FUNCTION_BLOCK TagCmp IMPLEMENTS I_TagCmp
VAR
	_iBaseTag		: I_Tag;
	_eResult		: Results.Result;
	_bLock			: BOOL;
END_VAR

PROPERTY PRIVATE _self : I_TagCmp
GET
VAR
	_this : I_TagCmp := THIS^;
END_VAR
_self := _this;
END_GET
END_PROPERTY

METHOD AndHasOption : I_TagCmp
VAR_INPUT
	sOption		: Strings.Str;
END_VAR
AndHasOption := _self;
sOption := Tc2_Utilities.F_ToLCase(sOption);

IF _bLock THEN
	RETURN;
END_IF

CASE _eResult OF
	Results.Ok,
	Results.None:
		IF _eResult = Results.Ok AND_THEN sOption <> '' AND_THEN _iBaseTag.Option = sOption THEN
			_eResult := Results.Ok;
		END_IF
END_CASE
END_METHOD

METHOD AndIf : I_TagCmp
VAR_INPUT
	bCondition: BOOL;
END_VAR
AndIf := _self;

IF _bLock THEN
	RETURN;
END_IF

IF _eResult = Results.Ok AND_THEN bCondition THEN
	_eResult := Results.Ok;
END_IF
END_METHOD

METHOD HasOption : I_TagCmp
VAR_INPUT
	sOption		: Strings.Str;
END_VAR
HasOption := _self;
sOption := Tc2_Utilities.F_ToLCase(sOption);

IF _bLock THEN
	RETURN;
END_IF

CASE _eResult OF
	Results.Ok,
	Results.None:
		IF sOption <> '' AND_THEN _iBaseTag.Option = sOption THEN
			_eResult := Results.Ok;
		END_IF
END_CASE
END_METHOD

METHOD IsErr : BOOL
IF _bLock THEN
	RETURN;
END_IF

IF _eResult >= 0 THEN
	RETURN;
END_IF

_bLock := TRUE;
IsErr := TRUE;
END_METHOD

METHOD IsFalse : BOOL
IF _bLock THEN
	RETURN;
END_IF

IF _eResult <> Results.None THEN
	RETURN;
END_IF

_bLock := TRUE;
IsFalse := TRUE;
END_METHOD

METHOD IsTrue : BOOL
IF _bLock THEN
	RETURN;
END_IF

IF _eResult <> Results.Ok THEN
	RETURN;
END_IF

_bLock := TRUE;
IsTrue := TRUE;
END_METHOD

METHOD Match : I_TagCmp
VAR_INPUT
	iOther: I_Tag;
END_VAR
Match := _self;

IF _bLock THEN
	RETURN;
END_IF

CASE _eResult OF
	Results.Ok,
	Results.None:
		IF iOther = _iBaseTag THEN
			_eResult := Results.Ok;
		END_IF
END_CASE
END_METHOD

METHOD MatchId : I_TagCmp
VAR_INPUT
	sIdToMatch		: Strings.Str;
END_VAR
MatchId := _self;
sIdToMatch := Tc2_Utilities.F_ToLCase(sIdToMatch);

IF _bLock THEN
	RETURN;
END_IF

CASE _eResult OF
	Results.Ok,
	Results.None:
		IF sIdToMatch <> '' AND_THEN (Tc2_Standard.RIGHT(_iBaseTag.GetId(), Tc2_Standard.LEN(sIdToMatch)) = sIdToMatch) THEN
			_eResult := Results.Ok;
		END_IF
END_CASE
END_METHOD

METHOD MatchWcdId : I_TagCmp
VAR_INPUT
	sPattern 			: Strings.Str;  					// Pattern with wildcards
END_VAR
VAR
	pttPath				: Strings.SymbolPath;
	pttSeg				: Strings.Str;
	pttPeek				: Strings.Str;
	addPath				: Strings.SymbolPath;
	addSeg				: Strings.Str;
END_VAR
MatchWcdId := _self;

// Check lock
IF _bLock THEN
	RETURN;
END_IF

// Check result state
CASE _eResult OF
	Results.Ok,
	Results.None:
		pttPath.Set(sPattern);
		addPath.Set(_iBaseTag.GetId());
		WHILE Results.IsOk(pttPath.Next(sSeg => pttSeg)) DO
		
			IF pttSeg = '*' THEN
				IF Results.IsOk(pttPath.Peek(sSeg => pttPeek)) THEN
					IF pttPeek = '*' THEN
						CONTINUE; // Skip redundant wildcard
					END_IF
				ELSE
					RETURN; // No more segments in the pattern, so it's a match
				END_IF
	
			ELSIF pttSeg <> '*' THEN
				pttPeek := '';
			END_IF
			
			WHILE Results.IsOk(addPath.Next(sSeg => addSeg)) DO
				IF pttPeek <> '' THEN
					IF pttPeek = addSeg THEN
						pttPath.Next();
						EXIT;
					ELSE
						CONTINUE;
					END_IF
				ELSIF pttSeg = addSeg THEN
					EXIT;
				ELSE
					RETURN;
				END_IF
			END_WHILE		
		END_WHILE
		
		IF Results.IsOk(addPath.Peek()) THEN
			RETURN;
		END_IF
		
		_eResult := Results.Ok;
END_CASE
END_METHOD

METHOD OrIf : I_TagCmp
VAR_INPUT
	bCondition: BOOL;
END_VAR
OrIf := _self;

IF _bLock THEN
	RETURN;
END_IF

IF _eResult = Results.Ok OR_ELSE bCondition THEN
	_eResult := Results.Ok;
END_IF
END_METHOD

METHOD Set : I_TagCmp
VAR_INPUT
	iBaseTag	: I_Tag;
END_VAR
_iBaseTag := iBaseTag;
_eResult := Results.None;
_bLock := FALSE;

IF iBaseTag = 0 THEN
	_eResult := Results.Err.Itf0;
END_IF

Set := _self;
END_METHOD

METHOD XorIf : I_TagCmp
VAR_INPUT
	bCondition: BOOL;
END_VAR
XorIf := _self;

IF _bLock THEN
	RETURN;
END_IF

IF _eResult = Results.Ok XOR bCondition THEN
	_eResult := Results.Ok;
END_IF
END_METHOD

END_FUNCTION_BLOCK

(* stored: Version 1.1.0.1
   POU TagCmp: Id {fc472a51-95c8-4c63-b8c5-5dfa13d61d73}, SpecialFunc None
   Property _self: Id {fe4340bb-7f6f-44d0-993a-3f0ac0014f79}
   Get Get: Id {e6bce7a1-dcf6-45e3-9283-e9e637ba0ada}
   Method AndHasOption: Id {4178bf0f-757c-43e4-9bd6-0c41f2c398f4}
   Method AndIf: Id {9223b46b-6be4-477a-9010-c0212fbeba73}
   Method HasOption: Id {c463345a-f124-40d6-b1f7-85e8eeaaf583}
   Method IsErr: Id {248d90f2-753e-444d-9c5b-49d2b4aa255c}
   Method IsFalse: Id {4388843a-3f13-4d13-9444-a6c347a1b77c}
   Method IsTrue: Id {866e2e11-40a2-444c-9771-a238b0485540}
   Method Match: Id {5c938a28-c260-4bf1-adcc-c84d59421fa8}
   Method MatchId: Id {78d82c00-f656-4a95-b467-0eabd905f45b}
   Method MatchWcdId: Id {155a5479-46da-4d47-bd5a-a8dff579e9de}
   Method OrIf: Id {c9bdb97c-3eb5-4133-8ad4-a1531337cf33}
   Method Set: Id {2167daab-4164-44b9-93b7-a85c88a05ebd}
   Method XorIf: Id {ca9c46ad-c94a-433e-aeab-483b4c5ea474} *)
